(* CODESYS project OMAC_PackML_State_Machine.library
   Description: The library ‘OMAC PackML State Machine’ contains a state machine for packaging controls based on the OMAC PackML standard.
      
      PackML, which stands for Packaging Machine Language, defines a common approach, or machine language, for automated machines. The primary goals are to encourage a common "look and feel" across a plant floor and to enable and encourage industry innovation.
      This library contains an implementation of the OMAC PackML State Machine. An example project shows the usage of the components. 
      For more information about OMAC and PackML see www.omac.org.
      
      The ‘PackML State Machine’ defines machine states and state transitions for packaging controls. A set of machines states is called ‘unit mode’. A unit mode can contain a maximum of 17 machine states. The following graphic shows all machine states with the corresponding state transitions.
      
      .. _figure1:
      
      .. figure:: ../Images/PackMLStates.png
      Figure 1: State transitions of PackML
      
      
      A machine state defines the current condition of a machine.  Three machine state types are proposed: 
       - Acting State (green), which was previously a Transient State, is one which represents some processing activity, i.e. STARTING, HOLDING,
       - Wait State (olive green), which was previously a Quiescent, or Steady State, is used to identify that a machine has achieved a defined set of conditions, i.e. ABORTED, HELD, SUSPENDED, IDLE.
       - Dual State (blue) is defined as wait state that is causing the machine to appear as an acting state. There is currently only one dual state: EXECUTE.
      
      A state transition is executed by a corresponding command like ‘Start’ or ‘Stop’.
      
      PackML allows to define own unit modes. For example it is possible to create own unit modes for setup or maintenance. The machine states of the defined unit modes are a subset of the 17 machine states.
      There is only one active unit mode allowed, but it is possible to switch between unit modes. This is handled by a component called unit mode manager. Before the unit mode will be switched, the unit mode manger checks if the current machine state allows leaving and if the target state allows entering.  
      
      .. _figure2:
      
      .. figure:: ../Images/UnitModeTransitions.png
      Figure 2: Unit mode transitions (© OMAC PackML Definiton Document V3.0) 
       
      Library OMAC_PackML_State_Machine
      ---------------------------------------------
      The package contains a library named ``OMAC_PackML_State_Machine`` which includes all required components to build a state machine based on PackML. 
      Unit modes can be defined with the function block |UnitMode|. The desired machine states can be set by the input field ``dwSupportedStates``. The permissions to switch between unit modes are handled by the input fields ``dwAllowsLeavingFromStates`` and ``dwAllowsEnteringIntoStates``. The machine state can be changed by calling the corresponding method in folder ``Commands`` (``Start, Stop, Abort…``).
      The function block |UnitModeManager| enables the switching of unit modes. All unit modes and the current state are managed by this function block.  
      
      
      Example project PackML_Example
      ----------------------------------------
      The project ``PackML_Example`` in the installation folder of the package includes two example applications with implemented PackML state machines.
      
      
      Application PackMLUnitModeManager
      ======================
      The application shows how to define own unit modes. The program ``PLC_PROG`` defines three unit modes (Production, Semi Auto and Setup). At first the unit modes must be registered at the |UnitModeManager|. After that, the current machine state and the current unit mode can be requested via the |UnitModeManager|. The current machine state and current unit mode are displayed by visualization.
      
      .. _figure3:
      
      .. figure:: ../Images/PackML.png
      Figure 3: Visualization of the application PackMLUnitModeManager
      
      
      Application PackMLAxisControl
      ==================
      The application ``PackMLAxisControl`` shows how to set the execution state of a virtual SoftMotion axis via the PackML state machine. The function block ``AxisControl`` represents an axis, which is controlled according to its active unit mode.
      
       .. _figure4:
      
      .. figure:: ../Images/PackML2.png
      Figure 4: Visualization of the application PackMLAxisControl
   Author: 3S - Smart Software Solutions GmbH
   Version: 1.0.0.4
   Company: 3S - Smart Software Solutions GmbH
   Title: OMAC PackML State Machine
   Placeholder: OMAC_PackML_State_Machine
   LanguageModelAttribute: qualified-access-only
   DefaultNamespace: PACK_ML
   DocFormat: reStructuredText

Project tree, tasks and I/O mapping:
  text list GlobalTextList
  OMAC_PackML_State_Machine/
    Function Blocks/
      function block UnitMode [ST]: Abort, ActingStateCompleted, Clear, Hold, Reset, Start, Stop, Suspend, UnHold, UnSuspend, CurrentState, Active, AllowsEntering, AllowsLeaving, Enter, NextState, Name, SupportedStates
      function block UnitModeManager [ST]: ActiveUnitMode, ActiveUnitModeNumber, AllowsSwitchingTo, FindMode, Register, SwitchUnitMode
    Visualization/
      visualisation UnitMode
    GlobalConstants/
      global variables GVL
    Enums/
      data type State
    Interfaces/
      interface IUnitMode: Abort, ActingStateCompleted, Clear, Hold, Reset, Start, Stop, Suspend, Unhold, UnSuspend, CurrentState, Name, SupportedStates, Active, AllowsEntering, AllowsLeaving, Enter, NextState
    image pool ImagePool
  00000000-0000-0000-0000-000000000000|D:\CoDeSys\LibrariesV3\trunk\Intern\CAA\CAA Template\3.4.0.0 draft\Placeholder.xml
  00000000-0000-0000-0000-000000000000|D:\CoDeSys\LibrariesV3\trunk\Intern\CAA\CAA Template\3.2.0.3 draft\Prefix.pdf
  00000000-0000-0000-0000-000000000000|D:\CoDeSys\LibrariesV3\trunk\Intern\CAA\CAA Template\3.5.2.0 draft\Placeholder.xml
  Images/
    PackML
    PackML2
    PackMLStates
    UnitModeTransitions
  5ce3da45-db07-42e7-a21c-a00fff4ed8f6|C:\Users\a.werner\Documents\background.jpg
*)

// OMAC_PackML_State_Machine/Enums/State
// Machine states
TYPE State :
(
	Stopped := 16#1, // Bit 0
	Resetting := 16#2, // Bit 1
	Idle := 16#4, // Bit 2
	Starting := 16#8, // Bit 3
	Execute := 16#10, // Bit 4
	Holding := 16#20, // Bit 5
	Held := 16#40, // Bit 6
	UnHolding := 16#80, // Bit 7
	Suspending := 16#100, // Bit 8
	Suspended := 16#200, // Bit 9
	UnSuspending := 16#400, // Bit 10
	Completing := 16#800, // Bit 11
	Complete := 16#1000, // Bit 12
	Stopping := 16#2000, // Bit 13
	Aborting := 16#4000, // Bit 14
	Aborted := 16#8000, // Bit 15
	Clearing := 16#10000, // Bit 16
	
	No := 0,
	All := 16#1FFFF,
	Invalid := 16#80000000
) DWORD;
END_TYPE

// OMAC_PackML_State_Machine/GlobalConstants/GVL
VAR_GLOBAL CONSTANT
	gc_usiMaxModes: USINT := 10;	// Maximum number of unit modes.
END_VAR

// OMAC_PackML_State_Machine/Function Blocks/UnitMode
// This function block describes an unit mode with all possible machine states, actions and the current state. 
// The transition between unit modes is handled by the UnitModeMangager. 
{attribute 'hide_all_locals'} 
FUNCTION_BLOCK UnitMode IMPLEMENTS IUnitMode
VAR_INPUT
	sName : STRING; // Name of the unit mode
	dwSupportedStates : DWORD := 2#11111111111111111; // Supported states
	dwAllowsLeavingFromStates : DWORD := State.Stopped OR State.Aborted; // Leaving state conditions
	dwAllowsEnteringIntoStates: DWORD := State.Stopped OR State.Aborted; // Entering state conditions
	eInitialState: State; // Initialization state
	xActive : BOOL; // True if this unit mode is active
END_VAR
VAR_OUTPUT
END_VAR
VAR
	eState:State:=State.Invalid;
	bInit: BOOL;
END_VAR

IF NOT bInit THEN
	bInit:=TRUE;
	eState := eInitialState;
END_IF

METHOD Abort : BOOL
VAR_INPUT
END_VAR
CASE eState OF
State.Stopped,
State.Resetting,
State.Idle,
State.Starting,
State.Execute,
State.Holding,
State.Held,
State.UnHolding,
State.Suspending,
State.Suspended,
State.UnSuspending,
State.Completing,
State.Complete,
State.Stopping,
State.Clearing:
	IF (State.Aborting AND SupportedStates) = 0 THEN
		Abort := FALSE;
		RETURN;
	END_IF
	eState := State.Aborting;
	Abort := TRUE;
END_CASE
END_METHOD

// This method should be called by the program if an action has been finished.
METHOD ActingStateCompleted : BOOL
VAR_INPUT
END_VAR
CASE eState OF
State.Holding,
State.UnHolding,
State.Starting,
State.Completing,
State.Resetting,
State.UnSuspending,
State.Suspending,
State.Aborting,
State.Stopping,
State.Clearing:
	IF (NextState(eState) AND SupportedStates) = 0 THEN
		ActingStateCompleted := FALSE;
		RETURN;
	END_IF
	eState := NextState(eState);
	ActingStateCompleted := TRUE;
	
State.Execute:
	IF (State.Completing AND SupportedStates) = 0 THEN
		ActingStateCompleted := FALSE;
		RETURN;
	END_IF
	eState := State.Completing;
	ActingStateCompleted := TRUE;
END_CASE

IF eState = State.Invalid THEN
	ActingStateCompleted := FALSE;
END_IF
END_METHOD

METHOD Clear : BOOL
VAR_INPUT
END_VAR
CASE eState OF
State.Aborted:
	IF (State.Clearing AND SupportedStates) = 0 THEN
		Clear := FALSE;
		RETURN;
	END_IF
	eState := State.Clearing;
	Clear := TRUE;
END_CASE
END_METHOD

METHOD Hold : BOOL
VAR_INPUT
END_VAR
CASE eState OF
State.Execute:
	IF (State.Holding AND SupportedStates) = 0 THEN
		Hold := FALSE;
		RETURN;
	END_IF
	eState := State.Holding;
	Hold := TRUE;
END_CASE
END_METHOD

METHOD Reset : BOOL
VAR_INPUT
END_VAR
CASE eState OF
State.Complete,
State.Stopped:
	IF (State.Resetting AND SupportedStates) = 0 THEN
		Reset := FALSE;
		RETURN;
	END_IF
	eState := State.Resetting;
	Reset := TRUE;
END_CASE
END_METHOD

METHOD Start : BOOL
VAR_INPUT
END_VAR
CASE eState OF
State.Idle:
	IF (State.Starting AND SupportedStates) = 0 THEN
		Start := FALSE;
		RETURN;
	END_IF
	eState := State.Starting;
	Start := TRUE;
END_CASE
END_METHOD

METHOD Stop : BOOL
VAR_INPUT
END_VAR
CASE eState OF
State.Resetting,
State.Idle,
State.Starting,
State.Execute,
State.Holding,
State.Held,
State.UnHolding,
State.Suspending,
State.Suspended,
State.UnSuspending,
State.Completing,
State.Complete:
	IF (State.Stopping AND SupportedStates) = 0 THEN
		Stop := FALSE;
		RETURN;
	END_IF
	eState := State.Stopping;
	Stop := TRUE;
END_CASE
END_METHOD

METHOD Suspend : BOOL
VAR_INPUT
END_VAR
CASE eState OF
State.Execute:
	IF (State.Suspending AND SupportedStates) = 0 THEN
		Suspend := FALSE;
		RETURN;
	END_IF
	eState := State.Suspending;
	Suspend := TRUE;
END_CASE
END_METHOD

METHOD UnHold : BOOL
VAR_INPUT
END_VAR
CASE eState OF
State.Held:
	IF (State.UnHolding AND SupportedStates) = 0 THEN
		UnHold := FALSE;
		RETURN;
	END_IF
	eState := State.UnHolding;
	UnHold := TRUE;
END_CASE
END_METHOD

METHOD UnSuspend : BOOL
VAR_INPUT
END_VAR
CASE eState OF
State.Suspended:
	IF (State.UnSuspending AND SupportedStates) = 0 THEN
		UnSuspend := FALSE;
		RETURN;
	END_IF
	eState := State.UnSuspending;
	UnSuspend := TRUE;
END_CASE
END_METHOD

// Get the current machine state
PROPERTY CurrentState : State
GET
CurrentState := eState;
END_GET
END_PROPERTY

// True if this unit mode is active.
PROPERTY Active : BOOL
GET
Active := xActive;
END_GET
SET
xActive := Active;
END_SET
END_PROPERTY

// Checks if the state allows entering.
{attribute 'hide'} 
METHOD AllowsEntering : BOOL
VAR_INPUT
	e: State;
END_VAR
IF (e AND dwAllowsEnteringIntoStates) > 0 THEN
	AllowsEntering := TRUE;
END_IF
END_METHOD

// True if the current state of this unit mode allows to be leaved.
PROPERTY AllowsLeaving : BOOL
GET
IF (eState AND dwAllowsLeavingFromStates) > 0 THEN
	AllowsLeaving := TRUE;
END_IF
END_GET
END_PROPERTY

// Enters the state.
METHOD Enter : BOOL
VAR_INPUT
	e: State;
END_VAR
eState := e;
END_METHOD

// Get the next machine state without checking the supported states.
METHOD NextState : State
VAR_INPUT
	e: State;
END_VAR
CASE e OF
State.Stopped:
	NextState := State.Resetting;
State.Resetting:
	NextState := State.Idle;
State.Idle:
	NextState := State.Starting;
State.Starting:
	NextState := State.Execute;
State.Execute:
	NextState := State.Invalid;
State.Holding:
	NextState := State.Held;
State.Held:
	NextState := State.UnHolding;
State.UnHolding:
	NextState := State.Execute;
State.Suspending:
	NextState := State.Suspended;
State.Suspended:
	NextState := State.UnSuspending;
State.UnSuspending:
	NextState := State.Execute;
State.Completing:
	NextState := State.Complete;
State.Complete:
	NextState := State.Resetting;
State.Stopping:
	NextState := State.Stopped;
State.Aborting:
	NextState := State.Aborted;
State.Aborted:
	NextState := State.Clearing;
State.Clearing:
	NextState := State.Stopped;
END_CASE
END_METHOD

// Get the name of the unit mode
PROPERTY Name : String
GET
Name := sName;
END_GET
END_PROPERTY

// Get all supported states.
PROPERTY SupportedStates : DWORD
GET
SupportedStates := dwSupportedStates;
END_GET
END_PROPERTY

END_FUNCTION_BLOCK

// OMAC_PackML_State_Machine/Interfaces/IUnitMode
INTERFACE IUnitMode

METHOD Abort : BOOL
VAR_INPUT
END_VAR
END_METHOD

METHOD ActingStateCompleted : BOOL
VAR_INPUT
END_VAR
END_METHOD

METHOD Clear : BOOL
VAR_INPUT
END_VAR
END_METHOD

METHOD Hold : BOOL
VAR_INPUT
END_VAR
END_METHOD

METHOD Reset : BOOL
VAR_INPUT
END_VAR
END_METHOD

METHOD Start : BOOL
VAR_INPUT
END_VAR
END_METHOD

METHOD Stop : BOOL
VAR_INPUT
END_VAR
END_METHOD

METHOD Suspend : BOOL
VAR_INPUT
END_VAR
END_METHOD

METHOD Unhold : BOOL
VAR_INPUT
END_VAR
END_METHOD

METHOD UnSuspend : BOOL
VAR_INPUT
END_VAR
END_METHOD

PROPERTY CurrentState : State
GET
END_GET
END_PROPERTY

PROPERTY Name : String
GET
END_GET
END_PROPERTY

PROPERTY SupportedStates : DWORD
GET
END_GET
END_PROPERTY

PROPERTY Active : BOOL
SET
END_SET
GET
END_GET
END_PROPERTY

METHOD AllowsEntering : BOOL
VAR_INPUT
	e: State;
END_VAR
END_METHOD

PROPERTY AllowsLeaving : BOOL
GET
END_GET
END_PROPERTY

METHOD Enter : BOOL
VAR_INPUT
	e: State;
END_VAR
END_METHOD

METHOD NextState : State
VAR_INPUT
	e: State;
END_VAR
END_METHOD

END_INTERFACE

// OMAC_PackML_State_Machine/Function Blocks/UnitModeManager
// Function block to switch the current unit mode.
{attribute 'hide_all_locals'} 
FUNCTION_BLOCK UnitModeManager
VAR_INPUT
END_VAR
VAR_OUTPUT
END_VAR
VAR
	apum: ARRAY[1..gc_usiMaxModes] OF IUnitMode;
	usiNumberOfUMs : USINT := 0;
	usiActualUM: USINT;
END_VAR

// Get and set the active unit mode.
PROPERTY ActiveUnitMode : IUnitMode
GET
ActiveUnitMode := apum[usiActualUM];
END_GET
END_PROPERTY

{attribute 'monitoring':='variable'}
PROPERTY ActiveUnitModeNumber : USINT
GET
ActiveUnitModeNumber := usiActualUM;
END_GET
END_PROPERTY

// Checks if the current state allows switching the current unit mode.
{attribute 'hide'} 
METHOD PRIVATE AllowsSwitchingTo : BOOL
VAR_INPUT
	usi: USINT; // Unit mode to switch
END_VAR
IF usi=usiActualUM THEN
	AllowsSwitchingTo := TRUE;
ELSE
	AllowsSwitchingTo := apum[usiActualUM].AllowsLeaving AND apum[usi].AllowsEntering(ActiveUnitMode.CurrentState);
END_IF
END_METHOD

// Finds an unit mode by name.
{attribute 'hide'} 
METHOD PRIVATE FindMode : USINT
VAR_INPUT
	sName: STRING; // Name od the unit mode
END_VAR
VAR
	usi: USINT;
END_VAR
FOR usi := 1 TO usiNumberOfUMs DO
	IF sName = apum[usi].Name THEN
		FindMode := usi;
		RETURN;
	END_IF
END_FOR
FindMode := gc_usiMaxModes+1;
END_METHOD

// Registers an unit mode
METHOD Register : BOOL
VAR_INPUT
	pum: IUnitMode;
END_VAR
IF usiNumberOfUMs < gc_usiMaxModes THEN
	usiNumberOfUMs := usiNumberOfUMs + 1;
	apum[usiNumberOfUMs] := pum;
	IF usiActualUM = 0 THEN
		usiActualUM := 1;
		apum[usiNumberOfUMs].Active := TRUE;
	ELSE
		apum[usiNumberOfUMs].Active := FALSE;
	END_IF
	Register := TRUE;
END_IF
END_METHOD

// Switch to an other unit mode and check the permission.
// Returns true if switching is allowed, returns false if switching is forbidden.
METHOD SwitchUnitMode : BOOL
VAR_INPUT
	sNewModeName: STRING; // Name of the unit mode to switch
END_VAR
VAR
	pnew: POINTER TO UnitMode;
	usi: USINT;
END_VAR
usi := FindMode(sNewModeName);
SwitchUnitMode := FALSE;
IF usi>gc_usiMaxModes THEN
	RETURN;
END_IF

IF usi=usiActualUM THEN
	SwitchUnitMode := TRUE;
	RETURN;
END_IF

IF apum[usiActualUM].AllowsLeaving AND apum[usi].AllowsEntering(ActiveUnitMode.CurrentState) THEN
	apum[usi].Enter(ActiveUnitMode.CurrentState);
	apum[usiActualUM].Active := FALSE;
	apum[usi].Active := TRUE;
	usiActualUM := usi;
	SwitchUnitMode := TRUE;
END_IF
END_METHOD

END_FUNCTION_BLOCK

// OMAC_PackML_State_Machine/Visualization/UnitMode
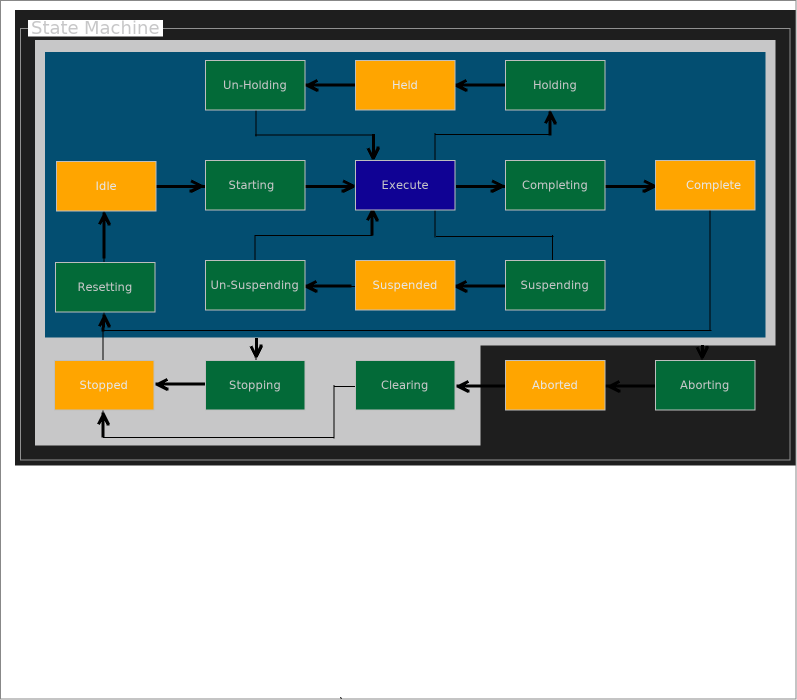
VISUALIZATION UnitMode  // 797x700
VAR_INPUT
	um: IUnitMode;
END_VAR
    Rectangle (15,10 780x455)
    GroupBox (20,20 770x440), "State Machine"
        Group (15,20 740x405)
            Polygon (0,0) (740,0) (740,305) (445,305) (445,405) (0,405)
            Rectangle (10,12 720x285)
            Polyline (149,146) (318,146) (308,151) (318,146) (308,141), invisible if: (um.SupportedStates AND State.Idle) = 0
            Polyline (69,218) (69,174) (74,184) (69,174) (64,184), invisible if: (um.SupportedStates AND State.Idle) = 0
            Line (69,275) (69,145), invisible if: (um.SupportedStates AND State.Idle) = 0
            Polyline (68,291) (69,276) (74,286) (69,276) (64,286), invisible if: (um.SupportedStates AND State.Complete) = 0 AND (um.SupportedStates AND State.Stopped) = 0
            Line (400,94) (516,94), invisible if: (um.SupportedStates AND State.Held) = 0
            Line (69,290) (676,290), invisible if: (um.SupportedStates AND State.Complete) = 0
            Line (299,398) (299,345), invisible if: (um.SupportedStates AND State.Aborted) = 0
            Line (299,346) (420,346), invisible if: (um.SupportedStates AND State.Aborted) = 0
            Polyline (573,346) (423,346) (433,351) (423,346) (433,341), invisible if: (um.SupportedStates AND State.Aborted) = 0
            Polyline (221,298) (221,316) (226,306) (221,316) (216,306), invisible if: (um.SupportedStates AND State.Stopped) = 0
            Line (221,345) (221,301), invisible if: (um.SupportedStates AND State.Stopped) = 0
            Polyline (668,346) (574,346) (584,351) (574,346) (584,341), invisible if: (um.SupportedStates AND State.Aborted) = 0
            Line (667,346) (667,306), invisible if: (um.SupportedStates AND State.Aborted) = 0
            Polyline (518,246) (421,246) (431,251) (421,246) (431,241), invisible if: (um.SupportedStates AND State.Suspended) = 0
            Polyline (667,305) (667,317) (672,307) (667,317) (662,307), invisible if: (um.SupportedStates AND State.Aborted) = 0
            Line (220,245) (220,195), invisible if: (um.SupportedStates AND State.Suspended) = 0
            Line (220,246) (421,246), invisible if: (um.SupportedStates AND State.Suspended) = 0
            Line (220,195) (337,195), invisible if: (um.SupportedStates AND State.Suspended) = 0
            Polyline (337,195) (337,170) (342,180) (337,170) (332,180), invisible if: (um.SupportedStates AND State.Suspended) = 0
            Polyline (316,246) (271,246) (281,251) (271,246) (281,241), invisible if: (um.SupportedStates AND State.Suspended) = 0
            Line (517,195) (517,248), invisible if: (um.SupportedStates AND State.Suspended) = 0
            Line (401,196) (518,196), invisible if: (um.SupportedStates AND State.Suspended) = 0
            Polyline (421,146) (467,146) (457,151) (467,146) (457,141), invisible if: (um.SupportedStates AND State.Complete) = 0
            Polyline (71,146) (166,146) (156,151) (166,146) (156,141), invisible if: (um.SupportedStates AND State.Idle) = 0
            Polyline (457,146) (619,146) (609,151) (619,146) (609,141), invisible if: (um.SupportedStates AND State.Complete) = 0
            Line (675,290) (675,145), invisible if: (um.SupportedStates AND State.Complete) = 0
            Line (527,146) (675,146), invisible if: (um.SupportedStates AND State.Complete) = 0
            Line (400,122) (400,93), invisible if: (um.SupportedStates AND State.Held) = 0
            Polyline (515,95) (515,73) (520,83) (515,73) (510,83), invisible if: (um.SupportedStates AND State.Held) = 0
            Line (338,95) (220,95), invisible if: (um.SupportedStates AND State.Held) = 0
            Polyline (338,94) (338,118) (343,108) (338,118) (333,108), invisible if: (um.SupportedStates AND State.Held) = 0
            Line (221,96) (221,43), invisible if: (um.SupportedStates AND State.Held) = 0
            Line (339,45) (221,45), invisible if: (um.SupportedStates AND State.Held) = 0
            Polyline (422,45) (272,45) (282,50) (272,45) (282,40), invisible if: (um.SupportedStates AND State.Held) = 0
            Line (515,94) (515,45), invisible if: (um.SupportedStates AND State.Held) = 0
            Polyline (516,45) (421,45) (431,50) (421,45) (431,40), invisible if: (um.SupportedStates AND State.Held) = 0
            Polygon (379,330) (381,326)
            Polyline (68,397) (68,374) (73,384) (68,374) (63,384), invisible if: (um.SupportedStates AND State.Aborted) = 0
            Line (68,397) (299,397), invisible if: (um.SupportedStates AND State.Aborted) = 0
            Line (400,197) (400,169), invisible if: (um.SupportedStates AND State.Suspended) = 0
            Line (68,319) (68,289), invisible if: (um.SupportedStates AND State.Complete) = 0 AND (um.SupportedStates AND State.Stopped) = 0
            Line (68,373) (68,318), invisible if: (um.SupportedStates AND State.Aborted) = 0
            RoundedRectangle (19,320 100x50), "Stopped", tooltip "The machine is stopped", colour toggle: um.CurrentState=State.Stopped, invisible if: (um.SupportedStates AND State.Stopped)=0
            RoundedRectangle (170,20 100x50), "Un-Holding", tooltip "The machine unholding to the Execute state", colour toggle: um.CurrentState=State.UnHolding, invisible if: (um.SupportedStates AND State.UnHolding)=0
            RoundedRectangle (320,120 100x50), "Execute", tooltip "The machine is executing the production logic", colour toggle: um.CurrentState=State.Execute, invisible if: (um.SupportedStates AND State.Execute)=0
            RoundedRectangle (20,222 100x50), "Resetting", tooltip "The machine resetting to the Idle state", colour toggle: um.CurrentState=State.Resetting, invisible if: (um.SupportedStates AND State.Resetting)=0
            RoundedRectangle (320,320 100x50), "Clearing", tooltip "The machine clearing from the Aborted state to the Stopped state", colour toggle: um.CurrentState=State.Clearing, invisible if: (um.SupportedStates AND State.Clearing)=0
            RoundedRectangle (470,320 100x50), "Aborted", tooltip "The machine is in the Aborted state", colour toggle: um.CurrentState=State.Aborted, invisible if: (um.SupportedStates AND State.Aborted)=0
            RoundedRectangle (620,320 100x50), "Aborting", tooltip "The machine is aborting to the Aborted state", colour toggle: um.CurrentState=State.Aborting, invisible if: (um.SupportedStates AND State.Aborting)=0
            RoundedRectangle (170,220 100x50), "Un-Suspending", tooltip "The machine unsuspending to the Execute state", colour toggle: um.CurrentState=State.UnSuspending, invisible if: (um.SupportedStates AND State.UnSuspending)=0
            RoundedRectangle (320,220 100x50), "Suspended", tooltip "The machine is suspended and waiting for an unsuspend command", colour toggle: um.CurrentState=State.Suspended, invisible if: (um.SupportedStates AND State.Suspended)=0
            RoundedRectangle (470,220 100x50), "Suspending", tooltip "The machine suspending to the Suspended state", colour toggle: um.CurrentState=State.Suspending, invisible if: (um.SupportedStates AND State.Suspending)=0
            RoundedRectangle (620,120 100x50), "Complete", tooltip "The machine has completed a production run and is waiting for a reset command", colour toggle: um.CurrentState=State.Complete, invisible if: (um.SupportedStates AND State.Complete)=0
            RoundedRectangle (470,120 100x50), "Completing", tooltip "The machine completing to the Complete state", colour toggle: um.CurrentState=State.Completing, invisible if: (um.SupportedStates AND State.Completing)=0
            RoundedRectangle (21,121 100x50), "Idle", tooltip "The machine is idle and waiting for a start command", colour toggle: um.CurrentState=State.Idle, invisible if: (um.SupportedStates AND State.Idle)=0
            RoundedRectangle (320,20 100x50), "Held", tooltip "The machine is held and waiting for an unhold command", colour toggle: um.CurrentState=State.Held, invisible if: (um.SupportedStates AND State.Held)=0
            RoundedRectangle (470,20 100x50), "Holding", tooltip "The machine holding to the Held state", colour toggle: um.CurrentState=State.Holding, invisible if: (um.SupportedStates AND State.Holding)=0
            Polyline (220,344) (122,344) (132,349) (122,344) (132,339), invisible if: (um.SupportedStates AND State.Stopped) = 0
            RoundedRectangle (170,120 100x50), "Starting", tooltip "The machine starting to the Execute state", colour toggle: um.CurrentState=State.Starting, invisible if: (um.SupportedStates AND State.Starting)=0
            RoundedRectangle (170,320 100x50), "Stopping", tooltip "The machine is stopping into the Stopped state", colour toggle: um.CurrentState=State.Stopping, invisible if: (um.SupportedStates AND State.Stopping)=0
    Polyline (340,697) (341,698)
END_VISUALIZATION
